// TIA Portal V17 export
// export: Created 2025-03-10T13:12:35.3649435Z, ExportSetting WithDefaults, DisplayName Totally Integrated Automation Portal, DisplayVersion V17 Update 8, DisplayName TIA Portal Openness, DisplayVersion V17 Update 8, DisplayName TIA Portal Version Control Interface, DisplayVersion V17, DisplayName SINAMICS Startdrive Advanced, DisplayVersion V17 SP2, DisplayName SINAMICS Startdrive G110M, G120, G120C, G120D, G120P, G115D, DisplayVersion V17 SP2, DisplayName SINAMICS Startdrive G130, G150, S120, S150, SINAMICS MV, S210, DisplayVersion V17 SP2, DisplayName STEP 7 Professional, DisplayVersion V17 Update 8, DisplayName SINUMERIK ONE STEP 7 Toolbox, DisplayVersion V17 Update 12, DisplayName SINUMERIK 840D sl STEP 7 Toolbox, DisplayVersion V17 Update 12, DisplayName STEP 7 Safety, DisplayVersion V17 Update 6, DisplayName WinCC Advanced, DisplayVersion V17 Update 8
FUNCTION "FC2103_ELECTRICAL_CABINET" : Void   // FC2103, LAD
{ S7_Optimized_Access := 'FALSE' }
AUTHOR : ETXETAR
VERSION : 1.0
// stored: AutoNumber false, IsIECCheckEnabled false, SetENOAutomatically false, UDAEnableTagReadback false
   VAR CONSTANT
      FC_NUMBER : DInt := 2103;
   END_VAR
   VAR_TEMP   // added for the SCL form of the ladder/FBD networks
      _w1 : Bool;
   END_VAR
BEGIN

REGION Network 1: INPUTS
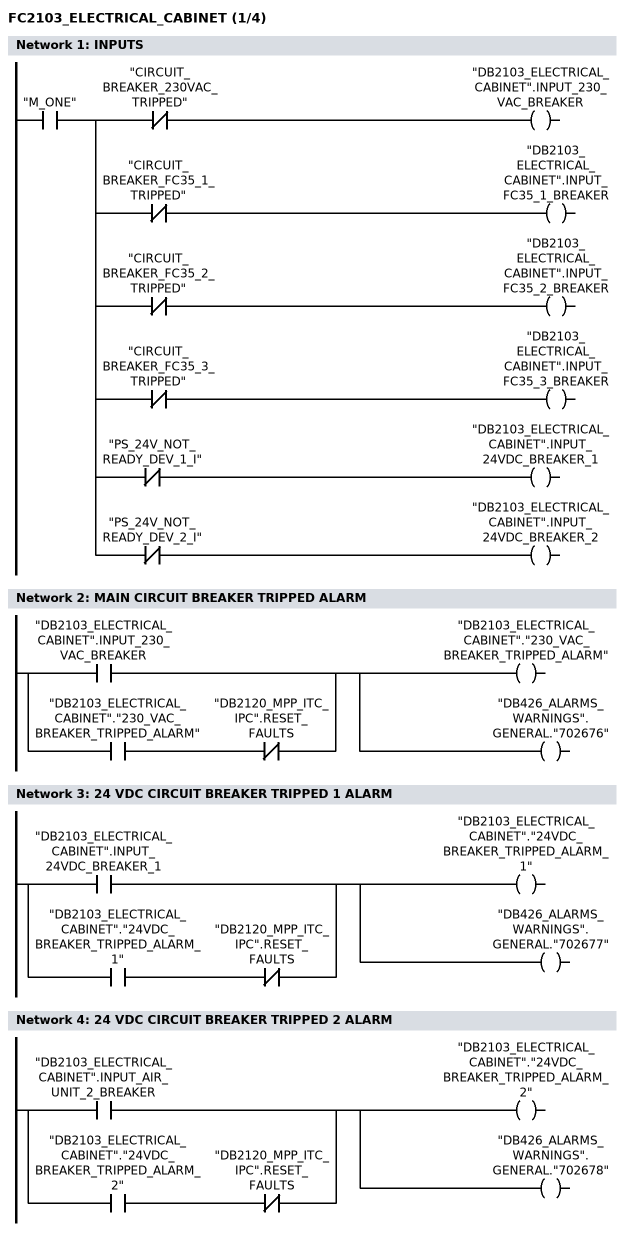
   RUNG wire#powerrail
      Contact( "M_ONE" )
      wire#w1
      I_Contact( "CIRCUIT_BREAKER_230VAC_TRIPPED" )
      Coil( "DB2103_ELECTRICAL_CABINET".INPUT_230_VAC_BREAKER )
   END_RUNG
   RUNG wire#w1
      I_Contact( "CIRCUIT_BREAKER_FC35_1_TRIPPED" )
      Coil( "DB2103_ELECTRICAL_CABINET".INPUT_FC35_1_BREAKER )
   END_RUNG
   RUNG wire#w1
      I_Contact( "CIRCUIT_BREAKER_FC35_2_TRIPPED" )
      Coil( "DB2103_ELECTRICAL_CABINET".INPUT_FC35_2_BREAKER )
   END_RUNG
   RUNG wire#w1
      I_Contact( "CIRCUIT_BREAKER_FC35_3_TRIPPED" )
      Coil( "DB2103_ELECTRICAL_CABINET".INPUT_FC35_3_BREAKER )
   END_RUNG
   RUNG wire#w1
      I_Contact( "PS_24V_NOT_READY_DEV_1_I" )
      Coil( "DB2103_ELECTRICAL_CABINET".INPUT_24VDC_BREAKER_1 )
   END_RUNG
   RUNG wire#w1
      I_Contact( "PS_24V_NOT_READY_DEV_2_I" )
      Coil( "DB2103_ELECTRICAL_CABINET".INPUT_24VDC_BREAKER_2 )
   END_RUNG
   // the same network as SCL:
   "DB2103_ELECTRICAL_CABINET".INPUT_230_VAC_BREAKER := "M_ONE" AND NOT "CIRCUIT_BREAKER_230VAC_TRIPPED";
   "DB2103_ELECTRICAL_CABINET".INPUT_FC35_1_BREAKER := "M_ONE" AND NOT "CIRCUIT_BREAKER_FC35_1_TRIPPED";
   "DB2103_ELECTRICAL_CABINET".INPUT_FC35_2_BREAKER := "M_ONE" AND NOT "CIRCUIT_BREAKER_FC35_2_TRIPPED";
   "DB2103_ELECTRICAL_CABINET".INPUT_FC35_3_BREAKER := "M_ONE" AND NOT "CIRCUIT_BREAKER_FC35_3_TRIPPED";
   "DB2103_ELECTRICAL_CABINET".INPUT_24VDC_BREAKER_1 := "M_ONE" AND NOT "PS_24V_NOT_READY_DEV_1_I";
   "DB2103_ELECTRICAL_CABINET".INPUT_24VDC_BREAKER_2 := "M_ONE" AND NOT "PS_24V_NOT_READY_DEV_2_I";
END_REGION

REGION Network 2: MAIN CIRCUIT BREAKER TRIPPED ALARM
   RUNG wire#powerrail
      Contact( "DB2103_ELECTRICAL_CABINET".INPUT_230_VAC_BREAKER )
      wire#w1
      Coil( "DB2103_ELECTRICAL_CABINET"."230_VAC_BREAKER_TRIPPED_ALARM" )
   END_RUNG
   RUNG wire#powerrail
      Contact( "DB2103_ELECTRICAL_CABINET"."230_VAC_BREAKER_TRIPPED_ALARM" )
      I_Contact( "DB2120_MPP_ITC_IPC".RESET_FAULTS )
   END_RUNG wire#w1
   RUNG wire#w1
      Coil( "DB426_ALARMS_WARNINGS".GENERAL."702676" )
   END_RUNG
   // the same network as SCL:
   "DB2103_ELECTRICAL_CABINET"."230_VAC_BREAKER_TRIPPED_ALARM" := "DB2103_ELECTRICAL_CABINET".INPUT_230_VAC_BREAKER OR ("DB2103_ELECTRICAL_CABINET"."230_VAC_BREAKER_TRIPPED_ALARM" AND NOT "DB2120_MPP_ITC_IPC".RESET_FAULTS);
   "DB426_ALARMS_WARNINGS".GENERAL."702676" := "DB2103_ELECTRICAL_CABINET"."230_VAC_BREAKER_TRIPPED_ALARM";
END_REGION

REGION Network 3: 24 VDC CIRCUIT BREAKER TRIPPED 1 ALARM
   RUNG wire#powerrail
      Contact( "DB2103_ELECTRICAL_CABINET".INPUT_24VDC_BREAKER_1 )
      wire#w1
      Coil( "DB2103_ELECTRICAL_CABINET"."24VDC_BREAKER_TRIPPED_ALARM_1" )
   END_RUNG
   RUNG wire#powerrail
      Contact( "DB2103_ELECTRICAL_CABINET"."24VDC_BREAKER_TRIPPED_ALARM_1" )
      I_Contact( "DB2120_MPP_ITC_IPC".RESET_FAULTS )
   END_RUNG wire#w1
   RUNG wire#w1
      Coil( "DB426_ALARMS_WARNINGS".GENERAL."702677" )
   END_RUNG
   // the same network as SCL:
   "DB2103_ELECTRICAL_CABINET"."24VDC_BREAKER_TRIPPED_ALARM_1" := "DB2103_ELECTRICAL_CABINET".INPUT_24VDC_BREAKER_1 OR ("DB2103_ELECTRICAL_CABINET"."24VDC_BREAKER_TRIPPED_ALARM_1" AND NOT "DB2120_MPP_ITC_IPC".RESET_FAULTS);
   "DB426_ALARMS_WARNINGS".GENERAL."702677" := "DB2103_ELECTRICAL_CABINET"."24VDC_BREAKER_TRIPPED_ALARM_1";
END_REGION

REGION Network 4: 24 VDC CIRCUIT BREAKER TRIPPED 2 ALARM
   RUNG wire#powerrail
      Contact( "DB2103_ELECTRICAL_CABINET".INPUT_AIR_UNIT_2_BREAKER )
      wire#w1
      Coil( "DB2103_ELECTRICAL_CABINET"."24VDC_BREAKER_TRIPPED_ALARM_2" )
   END_RUNG
   RUNG wire#powerrail
      Contact( "DB2103_ELECTRICAL_CABINET"."24VDC_BREAKER_TRIPPED_ALARM_2" )
      I_Contact( "DB2120_MPP_ITC_IPC".RESET_FAULTS )
   END_RUNG wire#w1
   RUNG wire#w1
      Coil( "DB426_ALARMS_WARNINGS".GENERAL."702678" )
   END_RUNG
   // the same network as SCL:
   "DB2103_ELECTRICAL_CABINET"."24VDC_BREAKER_TRIPPED_ALARM_2" := "DB2103_ELECTRICAL_CABINET".INPUT_AIR_UNIT_2_BREAKER OR ("DB2103_ELECTRICAL_CABINET"."24VDC_BREAKER_TRIPPED_ALARM_2" AND NOT "DB2120_MPP_ITC_IPC".RESET_FAULTS);
   "DB426_ALARMS_WARNINGS".GENERAL."702678" := "DB2103_ELECTRICAL_CABINET"."24VDC_BREAKER_TRIPPED_ALARM_2";
END_REGION

REGION Network 5: FC35_1 CIRCUIT BREAKER TRIPPED ALARM
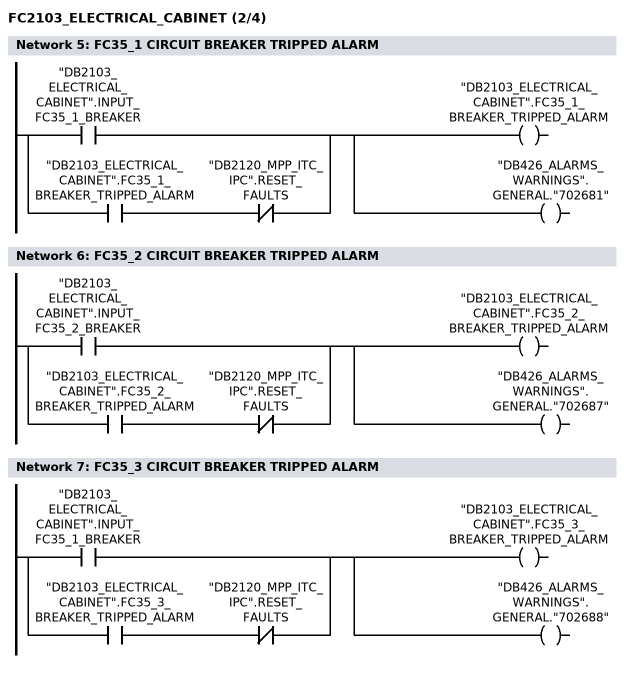
   RUNG wire#powerrail
      Contact( "DB2103_ELECTRICAL_CABINET".INPUT_FC35_1_BREAKER )
      wire#w1
      Coil( "DB2103_ELECTRICAL_CABINET".FC35_1_BREAKER_TRIPPED_ALARM )
   END_RUNG
   RUNG wire#powerrail
      Contact( "DB2103_ELECTRICAL_CABINET".FC35_1_BREAKER_TRIPPED_ALARM )
      I_Contact( "DB2120_MPP_ITC_IPC".RESET_FAULTS )
   END_RUNG wire#w1
   RUNG wire#w1
      Coil( "DB426_ALARMS_WARNINGS".GENERAL."702681" )
   END_RUNG
   // the same network as SCL:
   "DB2103_ELECTRICAL_CABINET".FC35_1_BREAKER_TRIPPED_ALARM := "DB2103_ELECTRICAL_CABINET".INPUT_FC35_1_BREAKER OR ("DB2103_ELECTRICAL_CABINET".FC35_1_BREAKER_TRIPPED_ALARM AND NOT "DB2120_MPP_ITC_IPC".RESET_FAULTS);
   "DB426_ALARMS_WARNINGS".GENERAL."702681" := "DB2103_ELECTRICAL_CABINET".FC35_1_BREAKER_TRIPPED_ALARM;
END_REGION

REGION Network 6: FC35_2 CIRCUIT BREAKER TRIPPED ALARM
   RUNG wire#powerrail
      Contact( "DB2103_ELECTRICAL_CABINET".INPUT_FC35_2_BREAKER )
      wire#w1
      Coil( "DB2103_ELECTRICAL_CABINET".FC35_2_BREAKER_TRIPPED_ALARM )
   END_RUNG
   RUNG wire#powerrail
      Contact( "DB2103_ELECTRICAL_CABINET".FC35_2_BREAKER_TRIPPED_ALARM )
      I_Contact( "DB2120_MPP_ITC_IPC".RESET_FAULTS )
   END_RUNG wire#w1
   RUNG wire#w1
      Coil( "DB426_ALARMS_WARNINGS".GENERAL."702687" )
   END_RUNG
   // the same network as SCL:
   "DB2103_ELECTRICAL_CABINET".FC35_2_BREAKER_TRIPPED_ALARM := "DB2103_ELECTRICAL_CABINET".INPUT_FC35_2_BREAKER OR ("DB2103_ELECTRICAL_CABINET".FC35_2_BREAKER_TRIPPED_ALARM AND NOT "DB2120_MPP_ITC_IPC".RESET_FAULTS);
   "DB426_ALARMS_WARNINGS".GENERAL."702687" := "DB2103_ELECTRICAL_CABINET".FC35_2_BREAKER_TRIPPED_ALARM;
END_REGION

REGION Network 7: FC35_3 CIRCUIT BREAKER TRIPPED ALARM
   RUNG wire#powerrail
      Contact( "DB2103_ELECTRICAL_CABINET".INPUT_FC35_1_BREAKER )
      wire#w1
      Coil( "DB2103_ELECTRICAL_CABINET".FC35_3_BREAKER_TRIPPED_ALARM )
   END_RUNG
   RUNG wire#powerrail
      Contact( "DB2103_ELECTRICAL_CABINET".FC35_3_BREAKER_TRIPPED_ALARM )
      I_Contact( "DB2120_MPP_ITC_IPC".RESET_FAULTS )
   END_RUNG wire#w1
   RUNG wire#w1
      Coil( "DB426_ALARMS_WARNINGS".GENERAL."702688" )
   END_RUNG
   // the same network as SCL:
   "DB2103_ELECTRICAL_CABINET".FC35_3_BREAKER_TRIPPED_ALARM := "DB2103_ELECTRICAL_CABINET".INPUT_FC35_1_BREAKER OR ("DB2103_ELECTRICAL_CABINET".FC35_3_BREAKER_TRIPPED_ALARM AND NOT "DB2120_MPP_ITC_IPC".RESET_FAULTS);
   "DB426_ALARMS_WARNINGS".GENERAL."702688" := "DB2103_ELECTRICAL_CABINET".FC35_3_BREAKER_TRIPPED_ALARM;
END_REGION

REGION Network 8: IMMEDIATE STOP ALARMS
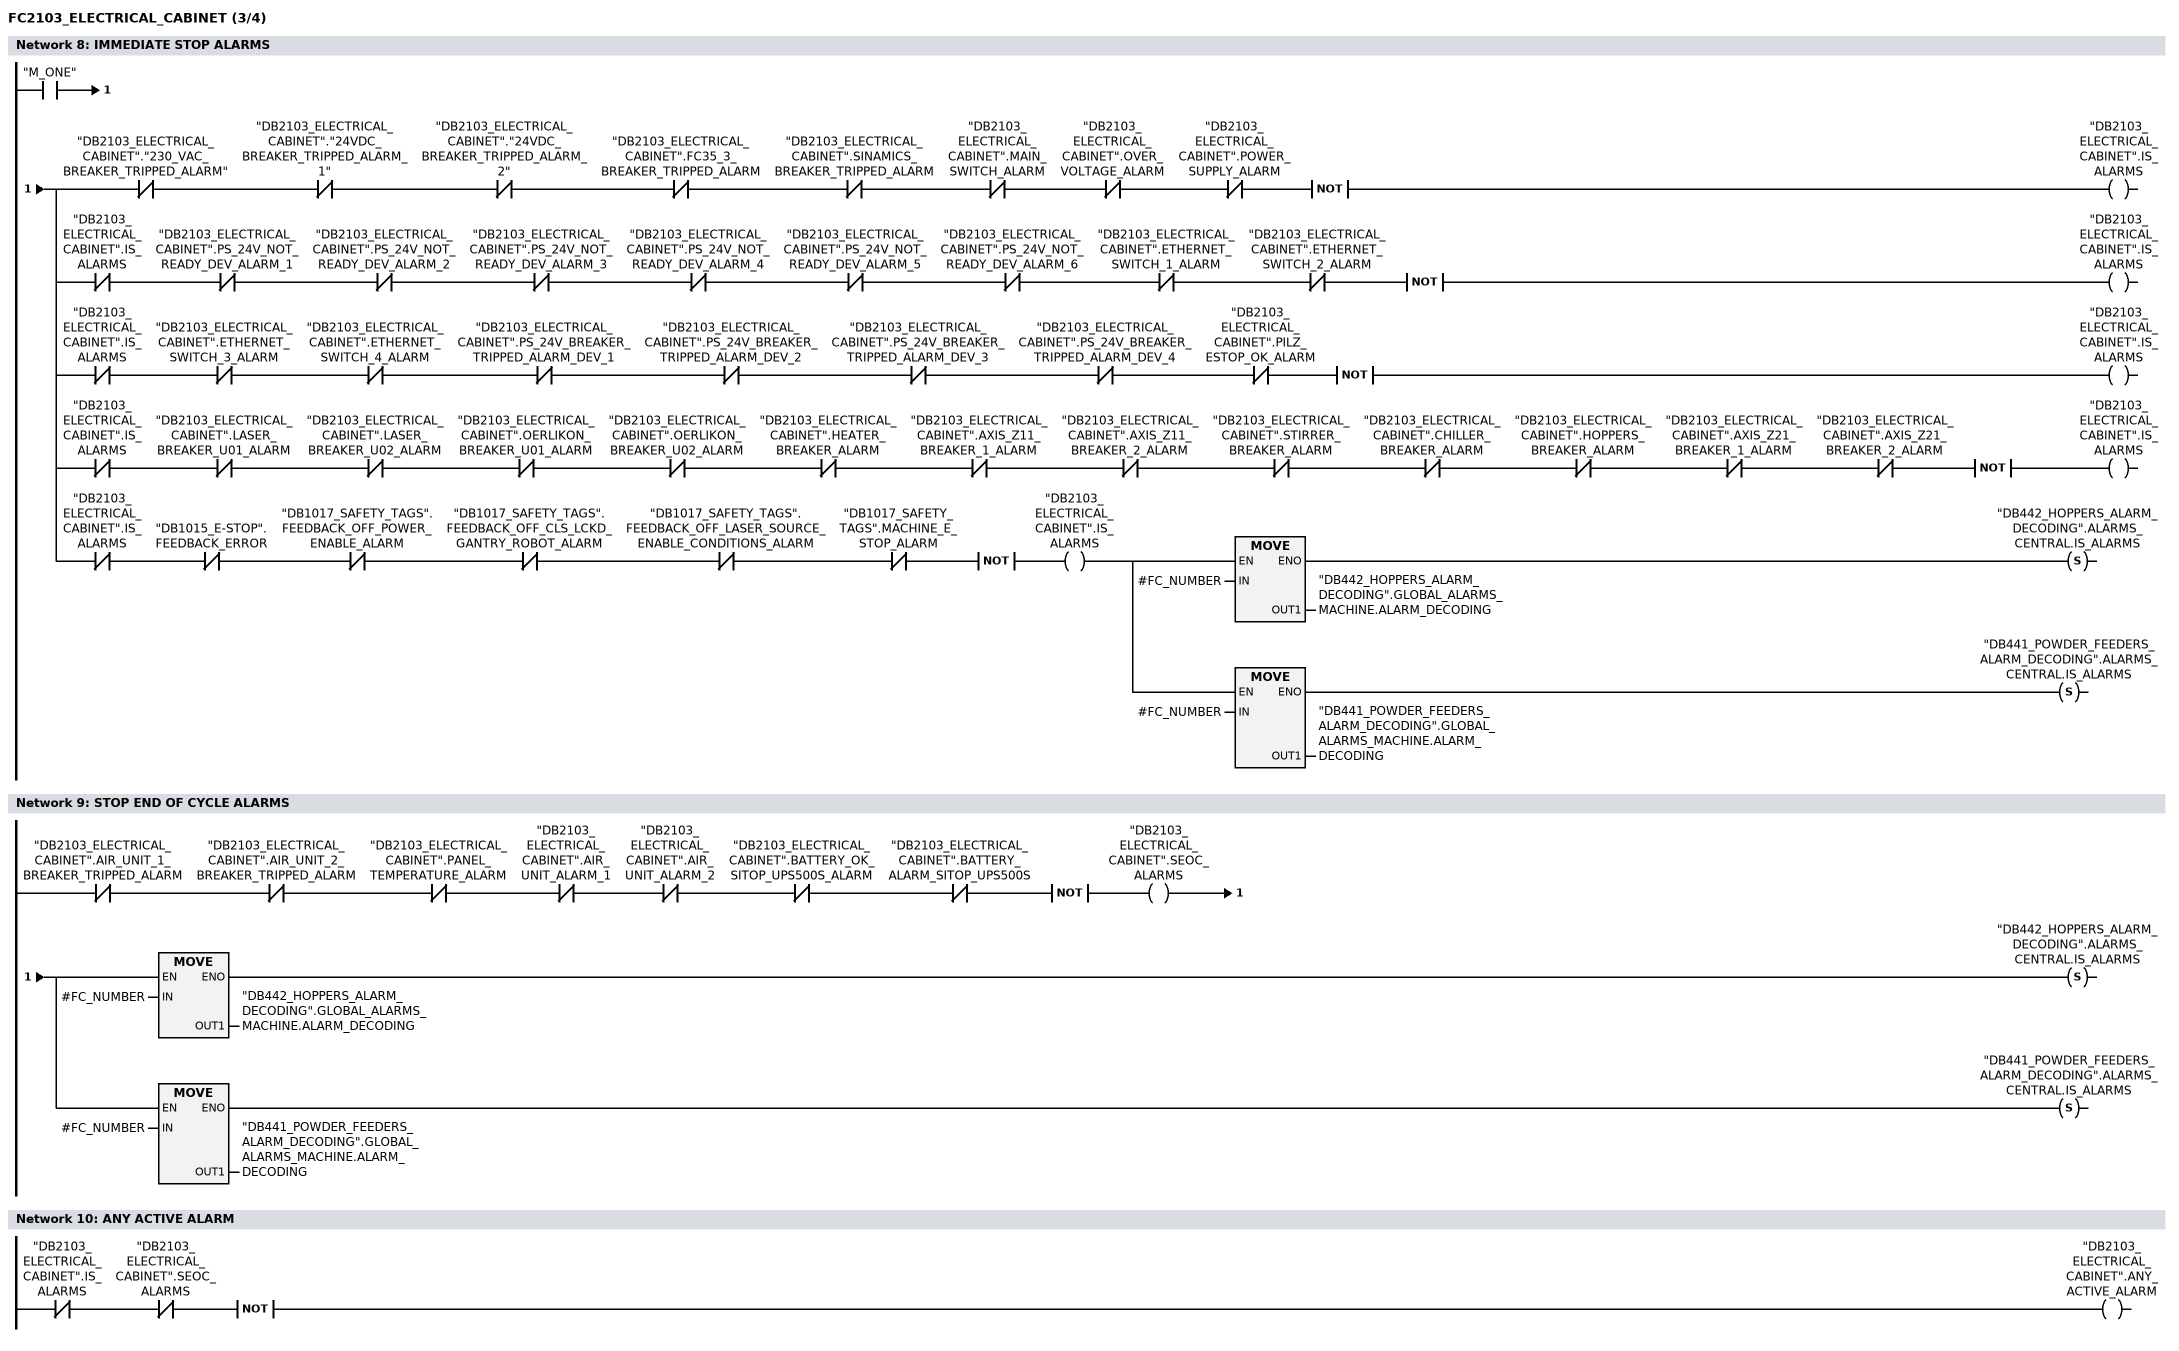
   RUNG wire#powerrail
      Contact( "M_ONE" )
      wire#w1
      I_Contact( "DB2103_ELECTRICAL_CABINET"."230_VAC_BREAKER_TRIPPED_ALARM" )
      I_Contact( "DB2103_ELECTRICAL_CABINET"."24VDC_BREAKER_TRIPPED_ALARM_1" )
      I_Contact( "DB2103_ELECTRICAL_CABINET"."24VDC_BREAKER_TRIPPED_ALARM_2" )
      I_Contact( "DB2103_ELECTRICAL_CABINET".FC35_3_BREAKER_TRIPPED_ALARM )
      I_Contact( "DB2103_ELECTRICAL_CABINET".SINAMICS_BREAKER_TRIPPED_ALARM )
      I_Contact( "DB2103_ELECTRICAL_CABINET".MAIN_SWITCH_ALARM )
      I_Contact( "DB2103_ELECTRICAL_CABINET".OVER_VOLTAGE_ALARM )
      I_Contact( "DB2103_ELECTRICAL_CABINET".POWER_SUPPLY_ALARM )
      Not()
      Coil( "DB2103_ELECTRICAL_CABINET".IS_ALARMS )
   END_RUNG
   RUNG wire#w1
      I_Contact( "DB2103_ELECTRICAL_CABINET".IS_ALARMS )
      I_Contact( "DB2103_ELECTRICAL_CABINET".PS_24V_NOT_READY_DEV_ALARM_1 )
      I_Contact( "DB2103_ELECTRICAL_CABINET".PS_24V_NOT_READY_DEV_ALARM_2 )
      I_Contact( "DB2103_ELECTRICAL_CABINET".PS_24V_NOT_READY_DEV_ALARM_3 )
      I_Contact( "DB2103_ELECTRICAL_CABINET".PS_24V_NOT_READY_DEV_ALARM_4 )
      I_Contact( "DB2103_ELECTRICAL_CABINET".PS_24V_NOT_READY_DEV_ALARM_5 )
      I_Contact( "DB2103_ELECTRICAL_CABINET".PS_24V_NOT_READY_DEV_ALARM_6 )
      I_Contact( "DB2103_ELECTRICAL_CABINET".ETHERNET_SWITCH_1_ALARM )
      I_Contact( "DB2103_ELECTRICAL_CABINET".ETHERNET_SWITCH_2_ALARM )
      Not()
      Coil( "DB2103_ELECTRICAL_CABINET".IS_ALARMS )
   END_RUNG
   RUNG wire#w1
      I_Contact( "DB2103_ELECTRICAL_CABINET".IS_ALARMS )
      I_Contact( "DB2103_ELECTRICAL_CABINET".ETHERNET_SWITCH_3_ALARM )
      I_Contact( "DB2103_ELECTRICAL_CABINET".ETHERNET_SWITCH_4_ALARM )
      I_Contact( "DB2103_ELECTRICAL_CABINET".PS_24V_BREAKER_TRIPPED_ALARM_DEV_1 )
      I_Contact( "DB2103_ELECTRICAL_CABINET".PS_24V_BREAKER_TRIPPED_ALARM_DEV_2 )
      I_Contact( "DB2103_ELECTRICAL_CABINET".PS_24V_BREAKER_TRIPPED_ALARM_DEV_3 )
      I_Contact( "DB2103_ELECTRICAL_CABINET".PS_24V_BREAKER_TRIPPED_ALARM_DEV_4 )
      I_Contact( "DB2103_ELECTRICAL_CABINET".PILZ_ESTOP_OK_ALARM )
      Not()
      Coil( "DB2103_ELECTRICAL_CABINET".IS_ALARMS )
   END_RUNG
   RUNG wire#w1
      I_Contact( "DB2103_ELECTRICAL_CABINET".IS_ALARMS )
      I_Contact( "DB2103_ELECTRICAL_CABINET".LASER_BREAKER_U01_ALARM )
      I_Contact( "DB2103_ELECTRICAL_CABINET".LASER_BREAKER_U02_ALARM )
      I_Contact( "DB2103_ELECTRICAL_CABINET".OERLIKON_BREAKER_U01_ALARM )
      I_Contact( "DB2103_ELECTRICAL_CABINET".OERLIKON_BREAKER_U02_ALARM )
      I_Contact( "DB2103_ELECTRICAL_CABINET".HEATER_BREAKER_ALARM )
      I_Contact( "DB2103_ELECTRICAL_CABINET".AXIS_Z11_BREAKER_1_ALARM )
      I_Contact( "DB2103_ELECTRICAL_CABINET".AXIS_Z11_BREAKER_2_ALARM )
      I_Contact( "DB2103_ELECTRICAL_CABINET".STIRRER_BREAKER_ALARM )
      I_Contact( "DB2103_ELECTRICAL_CABINET".CHILLER_BREAKER_ALARM )
      I_Contact( "DB2103_ELECTRICAL_CABINET".HOPPERS_BREAKER_ALARM )
      I_Contact( "DB2103_ELECTRICAL_CABINET".AXIS_Z21_BREAKER_1_ALARM )
      I_Contact( "DB2103_ELECTRICAL_CABINET".AXIS_Z21_BREAKER_2_ALARM )
      Not()
      Coil( "DB2103_ELECTRICAL_CABINET".IS_ALARMS )
   END_RUNG
   RUNG wire#w1
      I_Contact( "DB2103_ELECTRICAL_CABINET".IS_ALARMS )
      I_Contact( "DB1015_E-STOP".FEEDBACK_ERROR )
      I_Contact( "DB1017_SAFETY_TAGS".FEEDBACK_OFF_POWER_ENABLE_ALARM )
      I_Contact( "DB1017_SAFETY_TAGS".FEEDBACK_OFF_CLS_LCKD_GANTRY_ROBOT_ALARM )
      I_Contact( "DB1017_SAFETY_TAGS".FEEDBACK_OFF_LASER_SOURCE_ENABLE_CONDITIONS_ALARM )
      I_Contact( "DB1017_SAFETY_TAGS".MACHINE_E_STOP_ALARM )
      Not()
      Coil( "DB2103_ELECTRICAL_CABINET".IS_ALARMS )
      wire#w2
      { S7_GenerateENO := "TRUE" } Move(in := #FC_NUMBER, out1 => "DB442_HOPPERS_ALARM_DECODING".GLOBAL_ALARMS_MACHINE.ALARM_DECODING)
      S_Coil( "DB442_HOPPERS_ALARM_DECODING".ALARMS_CENTRAL.IS_ALARMS )
   END_RUNG
   RUNG wire#w2
      { S7_GenerateENO := "TRUE" } Move(in := #FC_NUMBER, out1 => "DB441_POWDER_FEEDERS_ALARM_DECODING".GLOBAL_ALARMS_MACHINE.ALARM_DECODING)
      S_Coil( "DB441_POWDER_FEEDERS_ALARM_DECODING".ALARMS_CENTRAL.IS_ALARMS )
   END_RUNG
   // the same network as SCL:
   // ENO of a box is taken as its EN; it also drops when the box reports an error
   "DB2103_ELECTRICAL_CABINET".IS_ALARMS := NOT ("M_ONE" AND NOT "DB2103_ELECTRICAL_CABINET"."230_VAC_BREAKER_TRIPPED_ALARM" AND NOT "DB2103_ELECTRICAL_CABINET"."24VDC_BREAKER_TRIPPED_ALARM_1" AND NOT "DB2103_ELECTRICAL_CABINET"."24VDC_BREAKER_TRIPPED_ALARM_2" AND NOT "DB2103_ELECTRICAL_CABINET".FC35_3_BREAKER_TRIPPED_ALARM AND NOT "DB2103_ELECTRICAL_CABINET".SINAMICS_BREAKER_TRIPPED_ALARM AND NOT "DB2103_ELECTRICAL_CABINET".MAIN_SWITCH_ALARM AND NOT "DB2103_ELECTRICAL_CABINET".OVER_VOLTAGE_ALARM AND NOT "DB2103_ELECTRICAL_CABINET".POWER_SUPPLY_ALARM);
   "DB2103_ELECTRICAL_CABINET".IS_ALARMS := NOT ("M_ONE" AND NOT "DB2103_ELECTRICAL_CABINET".IS_ALARMS AND NOT "DB2103_ELECTRICAL_CABINET".PS_24V_NOT_READY_DEV_ALARM_1 AND NOT "DB2103_ELECTRICAL_CABINET".PS_24V_NOT_READY_DEV_ALARM_2 AND NOT "DB2103_ELECTRICAL_CABINET".PS_24V_NOT_READY_DEV_ALARM_3 AND NOT "DB2103_ELECTRICAL_CABINET".PS_24V_NOT_READY_DEV_ALARM_4 AND NOT "DB2103_ELECTRICAL_CABINET".PS_24V_NOT_READY_DEV_ALARM_5 AND NOT "DB2103_ELECTRICAL_CABINET".PS_24V_NOT_READY_DEV_ALARM_6 AND NOT "DB2103_ELECTRICAL_CABINET".ETHERNET_SWITCH_1_ALARM AND NOT "DB2103_ELECTRICAL_CABINET".ETHERNET_SWITCH_2_ALARM);
   "DB2103_ELECTRICAL_CABINET".IS_ALARMS := NOT ("M_ONE" AND NOT "DB2103_ELECTRICAL_CABINET".IS_ALARMS AND NOT "DB2103_ELECTRICAL_CABINET".ETHERNET_SWITCH_3_ALARM AND NOT "DB2103_ELECTRICAL_CABINET".ETHERNET_SWITCH_4_ALARM AND NOT "DB2103_ELECTRICAL_CABINET".PS_24V_BREAKER_TRIPPED_ALARM_DEV_1 AND NOT "DB2103_ELECTRICAL_CABINET".PS_24V_BREAKER_TRIPPED_ALARM_DEV_2 AND NOT "DB2103_ELECTRICAL_CABINET".PS_24V_BREAKER_TRIPPED_ALARM_DEV_3 AND NOT "DB2103_ELECTRICAL_CABINET".PS_24V_BREAKER_TRIPPED_ALARM_DEV_4 AND NOT "DB2103_ELECTRICAL_CABINET".PILZ_ESTOP_OK_ALARM);
   "DB2103_ELECTRICAL_CABINET".IS_ALARMS := NOT ("M_ONE" AND NOT "DB2103_ELECTRICAL_CABINET".IS_ALARMS AND NOT "DB2103_ELECTRICAL_CABINET".LASER_BREAKER_U01_ALARM AND NOT "DB2103_ELECTRICAL_CABINET".LASER_BREAKER_U02_ALARM AND NOT "DB2103_ELECTRICAL_CABINET".OERLIKON_BREAKER_U01_ALARM AND NOT "DB2103_ELECTRICAL_CABINET".OERLIKON_BREAKER_U02_ALARM AND NOT "DB2103_ELECTRICAL_CABINET".HEATER_BREAKER_ALARM AND NOT "DB2103_ELECTRICAL_CABINET".AXIS_Z11_BREAKER_1_ALARM AND NOT "DB2103_ELECTRICAL_CABINET".AXIS_Z11_BREAKER_2_ALARM AND NOT "DB2103_ELECTRICAL_CABINET".STIRRER_BREAKER_ALARM AND NOT "DB2103_ELECTRICAL_CABINET".CHILLER_BREAKER_ALARM AND NOT "DB2103_ELECTRICAL_CABINET".HOPPERS_BREAKER_ALARM AND NOT "DB2103_ELECTRICAL_CABINET".AXIS_Z21_BREAKER_1_ALARM AND NOT "DB2103_ELECTRICAL_CABINET".AXIS_Z21_BREAKER_2_ALARM);
   "DB2103_ELECTRICAL_CABINET".IS_ALARMS := NOT ("M_ONE" AND NOT "DB2103_ELECTRICAL_CABINET".IS_ALARMS AND NOT "DB1015_E-STOP".FEEDBACK_ERROR AND NOT "DB1017_SAFETY_TAGS".FEEDBACK_OFF_POWER_ENABLE_ALARM AND NOT "DB1017_SAFETY_TAGS".FEEDBACK_OFF_CLS_LCKD_GANTRY_ROBOT_ALARM AND NOT "DB1017_SAFETY_TAGS".FEEDBACK_OFF_LASER_SOURCE_ENABLE_CONDITIONS_ALARM AND NOT "DB1017_SAFETY_TAGS".MACHINE_E_STOP_ALARM);
   IF "DB2103_ELECTRICAL_CABINET".IS_ALARMS THEN
       "DB442_HOPPERS_ALARM_DECODING".GLOBAL_ALARMS_MACHINE.ALARM_DECODING := #FC_NUMBER;
       "DB442_HOPPERS_ALARM_DECODING".ALARMS_CENTRAL.IS_ALARMS := TRUE;
       "DB441_POWDER_FEEDERS_ALARM_DECODING".GLOBAL_ALARMS_MACHINE.ALARM_DECODING := #FC_NUMBER;
       "DB441_POWDER_FEEDERS_ALARM_DECODING".ALARMS_CENTRAL.IS_ALARMS := TRUE;
   END_IF;
END_REGION

REGION Network 9: STOP END OF CYCLE ALARMS
   RUNG wire#powerrail
      I_Contact( "DB2103_ELECTRICAL_CABINET".AIR_UNIT_1_BREAKER_TRIPPED_ALARM )
      I_Contact( "DB2103_ELECTRICAL_CABINET".AIR_UNIT_2_BREAKER_TRIPPED_ALARM )
      I_Contact( "DB2103_ELECTRICAL_CABINET".PANEL_TEMPERATURE_ALARM )
      I_Contact( "DB2103_ELECTRICAL_CABINET".AIR_UNIT_ALARM_1 )
      I_Contact( "DB2103_ELECTRICAL_CABINET".AIR_UNIT_ALARM_2 )
      I_Contact( "DB2103_ELECTRICAL_CABINET".BATTERY_OK_SITOP_UPS500S_ALARM )
      I_Contact( "DB2103_ELECTRICAL_CABINET".BATTERY_ALARM_SITOP_UPS500S )
      Not()
      Coil( "DB2103_ELECTRICAL_CABINET".SEOC_ALARMS )
      wire#w1
      { S7_GenerateENO := "TRUE" } Move(in := #FC_NUMBER, out1 => "DB442_HOPPERS_ALARM_DECODING".GLOBAL_ALARMS_MACHINE.ALARM_DECODING)
      S_Coil( "DB442_HOPPERS_ALARM_DECODING".ALARMS_CENTRAL.IS_ALARMS )
   END_RUNG
   RUNG wire#w1
      { S7_GenerateENO := "TRUE" } Move(in := #FC_NUMBER, out1 => "DB441_POWDER_FEEDERS_ALARM_DECODING".GLOBAL_ALARMS_MACHINE.ALARM_DECODING)
      S_Coil( "DB441_POWDER_FEEDERS_ALARM_DECODING".ALARMS_CENTRAL.IS_ALARMS )
   END_RUNG
   // the same network as SCL:
   // ENO of a box is taken as its EN; it also drops when the box reports an error
   "DB2103_ELECTRICAL_CABINET".SEOC_ALARMS := NOT (NOT "DB2103_ELECTRICAL_CABINET".AIR_UNIT_1_BREAKER_TRIPPED_ALARM AND NOT "DB2103_ELECTRICAL_CABINET".AIR_UNIT_2_BREAKER_TRIPPED_ALARM AND NOT "DB2103_ELECTRICAL_CABINET".PANEL_TEMPERATURE_ALARM AND NOT "DB2103_ELECTRICAL_CABINET".AIR_UNIT_ALARM_1 AND NOT "DB2103_ELECTRICAL_CABINET".AIR_UNIT_ALARM_2 AND NOT "DB2103_ELECTRICAL_CABINET".BATTERY_OK_SITOP_UPS500S_ALARM AND NOT "DB2103_ELECTRICAL_CABINET".BATTERY_ALARM_SITOP_UPS500S);
   IF "DB2103_ELECTRICAL_CABINET".SEOC_ALARMS THEN
       "DB442_HOPPERS_ALARM_DECODING".GLOBAL_ALARMS_MACHINE.ALARM_DECODING := #FC_NUMBER;
       "DB442_HOPPERS_ALARM_DECODING".ALARMS_CENTRAL.IS_ALARMS := TRUE;
       "DB441_POWDER_FEEDERS_ALARM_DECODING".GLOBAL_ALARMS_MACHINE.ALARM_DECODING := #FC_NUMBER;
       "DB441_POWDER_FEEDERS_ALARM_DECODING".ALARMS_CENTRAL.IS_ALARMS := TRUE;
   END_IF;
END_REGION

REGION Network 10: ANY ACTIVE ALARM
   RUNG wire#powerrail
      I_Contact( "DB2103_ELECTRICAL_CABINET".IS_ALARMS )
      I_Contact( "DB2103_ELECTRICAL_CABINET".SEOC_ALARMS )
      Not()
      Coil( "DB2103_ELECTRICAL_CABINET".ANY_ACTIVE_ALARM )
   END_RUNG
   // the same network as SCL:
   "DB2103_ELECTRICAL_CABINET".ANY_ACTIVE_ALARM := NOT (NOT "DB2103_ELECTRICAL_CABINET".IS_ALARMS AND NOT "DB2103_ELECTRICAL_CABINET".SEOC_ALARMS);
END_REGION

REGION Network 11: WARNINGS
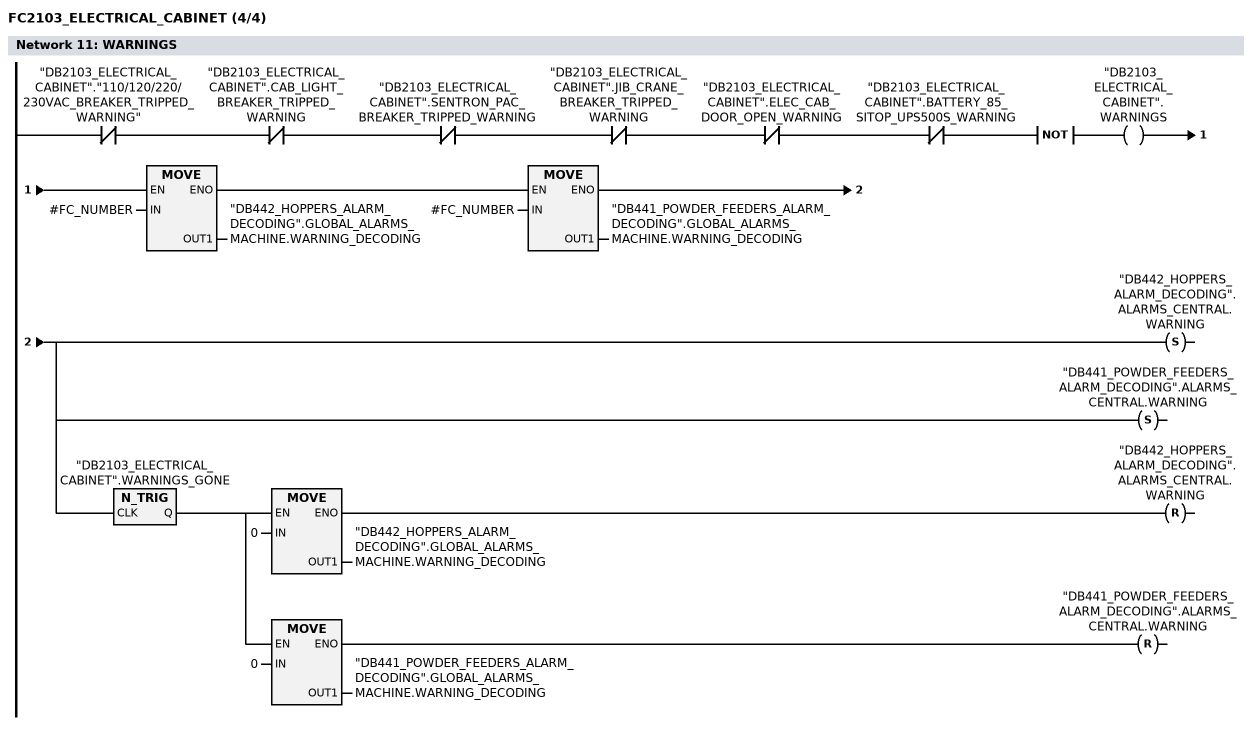
   RUNG wire#powerrail
      I_Contact( "DB2103_ELECTRICAL_CABINET"."110/120/220/230VAC_BREAKER_TRIPPED_WARNING" )
      I_Contact( "DB2103_ELECTRICAL_CABINET".CAB_LIGHT_BREAKER_TRIPPED_WARNING )
      I_Contact( "DB2103_ELECTRICAL_CABINET".SENTRON_PAC_BREAKER_TRIPPED_WARNING )
      I_Contact( "DB2103_ELECTRICAL_CABINET".JIB_CRANE_BREAKER_TRIPPED_WARNING )
      I_Contact( "DB2103_ELECTRICAL_CABINET".ELEC_CAB_DOOR_OPEN_WARNING )
      I_Contact( "DB2103_ELECTRICAL_CABINET".BATTERY_85_SITOP_UPS500S_WARNING )
      Not()
      Coil( "DB2103_ELECTRICAL_CABINET".WARNINGS )
      { S7_GenerateENO := "TRUE" } Move(in := #FC_NUMBER, out1 => "DB442_HOPPERS_ALARM_DECODING".GLOBAL_ALARMS_MACHINE.WARNING_DECODING)
      { S7_GenerateENO := "TRUE" } Move(in := #FC_NUMBER, out1 => "DB441_POWDER_FEEDERS_ALARM_DECODING".GLOBAL_ALARMS_MACHINE.WARNING_DECODING)
      wire#w1
      S_Coil( "DB442_HOPPERS_ALARM_DECODING".ALARMS_CENTRAL.WARNING )
   END_RUNG
   RUNG wire#w1
      S_Coil( "DB441_POWDER_FEEDERS_ALARM_DECODING".ALARMS_CENTRAL.WARNING )
   END_RUNG
   RUNG wire#w1
      N_Trig( "DB2103_ELECTRICAL_CABINET".WARNINGS_GONE )
      wire#w2
      { S7_GenerateENO := "TRUE" } Move(in := 0, out1 => "DB442_HOPPERS_ALARM_DECODING".GLOBAL_ALARMS_MACHINE.WARNING_DECODING)
      R_Coil( "DB442_HOPPERS_ALARM_DECODING".ALARMS_CENTRAL.WARNING )
   END_RUNG
   RUNG wire#w2
      { S7_GenerateENO := "TRUE" } Move(in := 0, out1 => "DB441_POWDER_FEEDERS_ALARM_DECODING".GLOBAL_ALARMS_MACHINE.WARNING_DECODING)
      R_Coil( "DB441_POWDER_FEEDERS_ALARM_DECODING".ALARMS_CENTRAL.WARNING )
   END_RUNG
   // the same network as SCL:
   // ENO of a box is taken as its EN; it also drops when the box reports an error
   "DB2103_ELECTRICAL_CABINET".WARNINGS := NOT (NOT "DB2103_ELECTRICAL_CABINET"."110/120/220/230VAC_BREAKER_TRIPPED_WARNING" AND NOT "DB2103_ELECTRICAL_CABINET".CAB_LIGHT_BREAKER_TRIPPED_WARNING AND NOT "DB2103_ELECTRICAL_CABINET".SENTRON_PAC_BREAKER_TRIPPED_WARNING AND NOT "DB2103_ELECTRICAL_CABINET".JIB_CRANE_BREAKER_TRIPPED_WARNING AND NOT "DB2103_ELECTRICAL_CABINET".ELEC_CAB_DOOR_OPEN_WARNING AND NOT "DB2103_ELECTRICAL_CABINET".BATTERY_85_SITOP_UPS500S_WARNING);
   IF "DB2103_ELECTRICAL_CABINET".WARNINGS THEN
       "DB442_HOPPERS_ALARM_DECODING".GLOBAL_ALARMS_MACHINE.WARNING_DECODING := #FC_NUMBER;
       "DB441_POWDER_FEEDERS_ALARM_DECODING".GLOBAL_ALARMS_MACHINE.WARNING_DECODING := #FC_NUMBER;
       "DB442_HOPPERS_ALARM_DECODING".ALARMS_CENTRAL.WARNING := TRUE;
       "DB441_POWDER_FEEDERS_ALARM_DECODING".ALARMS_CENTRAL.WARNING := TRUE;
   END_IF;
   #_w1 := NOT "DB2103_ELECTRICAL_CABINET".WARNINGS AND "DB2103_ELECTRICAL_CABINET".WARNINGS_GONE;   // falling edge
   "DB2103_ELECTRICAL_CABINET".WARNINGS_GONE := "DB2103_ELECTRICAL_CABINET".WARNINGS;
   IF #_w1 THEN
       "DB442_HOPPERS_ALARM_DECODING".GLOBAL_ALARMS_MACHINE.WARNING_DECODING := 0;
       "DB442_HOPPERS_ALARM_DECODING".ALARMS_CENTRAL.WARNING := FALSE;
       "DB441_POWDER_FEEDERS_ALARM_DECODING".GLOBAL_ALARMS_MACHINE.WARNING_DECODING := 0;
       "DB441_POWDER_FEEDERS_ALARM_DECODING".ALARMS_CENTRAL.WARNING := FALSE;
   END_IF;
END_REGION
END_FUNCTION
